# EPICS autosave request: profile_bluesky/startup/ref/Db/femtopd.req
$(P)$(H)$(F)vfc
$(P)$(H)$(F)mode
$(P)$(H)$(F)gain
$(P)$(H)$(F)gainU
$(P)$(H)$(F)gainD
$(P)$(H)$(F)gain0
$(P)$(H)$(F)gain1
$(P)$(H)$(F)gain2
$(P)$(H)$(F)gain3
$(P)$(H)$(F)gain4
$(P)$(H)$(F)bkg0
$(P)$(H)$(F)bkg1
$(P)$(H)$(F)bkg2
$(P)$(H)$(F)bkg3
$(P)$(H)$(F)bkg4
$(P)$(H)$(F)bkgErr0
$(P)$(H)$(F)bkgErr1
$(P)$(H)$(F)bkgErr2
$(P)$(H)$(F)bkgErr3
$(P)$(H)$(F)bkgErr4
$(P)$(H)$(F)reqrange
